// TIA Portal V18 export
FUNCTION "CuringOven" : Void   // FC900, LAD
{ S7_Optimized_Access := 'TRUE' }
// stored: AutoNumber false, SetENOAutomatically false
BEGIN

REGION Network 1
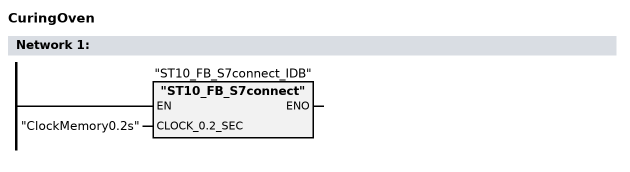
   RUNG wire#powerrail
      "ST10_FB_S7connect_IDB"("CLOCK_0.2_SEC" := "ClockMemory0.2s")
   END_RUNG
   // the same network as SCL:
   "ST10_FB_S7connect_IDB"("CLOCK_0.2_SEC" := "ClockMemory0.2s");   // "ST10_FB_S7connect"
END_REGION
END_FUNCTION
